// TIA Portal V15.1 export
// export: Created 2020-06-12T07:35:56.2568359Z, ExportSetting None, DisplayName Totally Integrated Automation Portal, DisplayVersion V15.1, DisplayName TIA Portal Openness, DisplayVersion V15.1, DisplayName STEP 7 Professional, DisplayVersion V15.1, DisplayName STEP 7 Safety, DisplayVersion V15.1, DisplayName WinCC Advanced, DisplayVersion V15.1
FUNCTION "SIM_PROC" : Void   // FC194, FBD
{ S7_Optimized_Access := 'TRUE' }
// stored: SetENOAutomatically False
   VAR_TEMP
      _cont_reset : Bool;
      _rVal : Real;
   END_VAR
BEGIN

REGION Network 1: TEST PID (0)
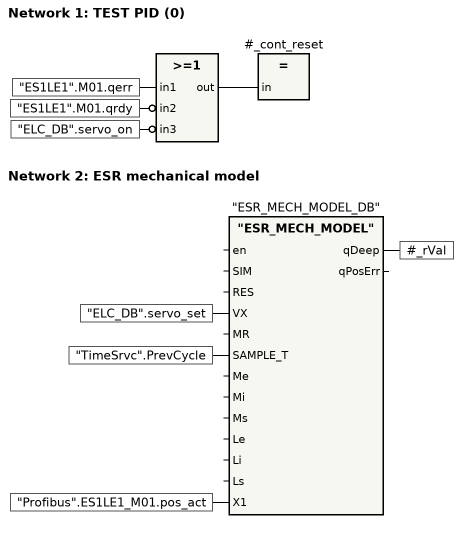
   #_cont_reset := "ES1LE1".M01.qerr OR NOT "ES1LE1".M01.qrdy OR NOT "ELC_DB".servo_on;
END_REGION

REGION Network 2: ESR mechanical model
   // X1(0) = 3950 mm
   "ESR_MECH_MODEL_DB"(VX := "ELC_DB".servo_set,   // "ESR_MECH_MODEL"
                       SAMPLE_T := "TimeSrvc".PrevCycle,
                       X1 := "Profibus".ES1LE1_M01.pos_act,
                       qDeep => #_rVal);
END_REGION
END_FUNCTION
